TYPE ST_SystemEval :
STRUCT
    bAllModulesOff : BOOL;
    bAnyModuleActive : BOOL;
    bAnyModuleFault : BOOL;
    bGridOk : BOOL;

    rTotalAvailableCurrent : REAL;
    rMaxTemperature : REAL;
    iHealthyModules : INT;
END_STRUCT
END_TYPE

(* stored: Version 1.1.0.1, ProductVersion 3.1.4026.18
   DUT ST_SystemEval: Id {a670cbad-400c-4c60-8a14-0c5231b2e5d4} *)
